TYPE BeltOut :
STRUCT
	belt : Belt;
	photo_sensor :ARRAY[0..2]OF BOOL;
END_STRUCT
END_TYPE

(* stored: Version 1.1.0.1, ProductVersion 3.1.4024.12
   DUT BeltOut: Id {c782cc16-e9cc-4232-8135-3777a46402f6} *)
